FUNCTION_BLOCK FB_TransportTube
VAR_INPUT
	i_stConfig : ST_TransportTubeConfig;
	i_bLaserExtIntl : BOOL; // external interlock for laser
END_VAR
VAR_OUTPUT	
	{attribute 'pytmc' := '
		pv: LASER_OK
		io: o
		field: ZNAM NOT_OK
		field: ONAM OK
	'}
	q_bLaserOk : BOOL; // Whether the laser is ok for operation
	
	{attribute 'pytmc' := '
		pv:
	'}
	q_stConfig : ST_TransportTubeConfig;
END_VAR
VAR
	bLaserOk : BOOL;
END_VAR

q_stConfig := i_stConfig;
q_bLaserOk := i_bLaserExtIntl AND bLaserOk;

METHOD PUBLIC M_SetLaserOk
VAR_INPUT
	i_bVal : BOOL;
END_VAR
bLaserOk := i_bVal;
END_METHOD

END_FUNCTION_BLOCK

(* stored: Version 1.1.0.1, ProductVersion 3.1.4022.17
   POU FB_TransportTube: Id {4b66ee4b-c91a-4936-b397-8ff461536138}, SpecialFunc None
   Method M_SetLaserOk: Id {edae87a2-aeaf-4afa-b84e-38dce6a2b658} *)
